// Mitsubishi GX Works2 project: GilKor   PLC: FX3G

// global labels: Global1
VAR_GLOBAL
  Switch7 AT X007 : BOOL;
  Lamp7 AT Y007 : BOOL;
END_VAR
VAR_GLOBAL CONSTANT
  Constant1 : BOOL := TRUE;
END_VAR
VAR_GLOBAL
  Switch1 AT X001 : BOOL;
  Switch2 AT X002 : BOOL;
  Lamp2 AT Y002 : BOOL;
  Lamp0 AT M1 : BOOL;
END_VAR

// task Task_01 (event TRUE, interval 0, priority 31): POU_01

PROGRAM POU_01
(* structured ladder/FBD written out as ST: instructions are called as NAME(EN, inputs, outputs); _pN, _eN, _tN stand for wires *)
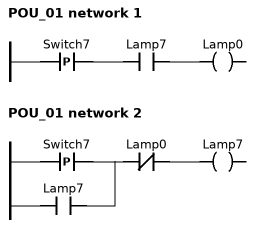
(* network 1 *)
Lamp0 := LDP(TRUE, Switch7) AND Lamp7;
(* network 2 *)
Lamp7 := (LDP(TRUE, Switch7) OR Lamp7) AND NOT Lamp0;
END_PROGRAM
